// TwinCAT 3 PLC project PayloadCarrier
// ProgramVersion: 3.1.4023.0
// libraries:
//   Tc2_Standard, * (Beckhoff Automation GmbH)
//   Tc2_System, * (Beckhoff Automation GmbH)
//   Tc3_Module, * (Beckhoff Automation GmbH)
// project tree:
//   DUTs/ E_PAYLOAD_CARRIER_MODE.TcDUT, E_Payload_Type.TcDUT, ST_SynchPayload.TcDUT
//   GVLs/ Global.TcGVL
//   / PlcTask.TcTTO
//   POUs/ A_Payload.TcPOU, I_Payload.TcIO, I_Payload_A.TcIO, I_Payload_B.TcIO, PayloadCarrier.TcPOU, Payload_A.TcPOU, MAIN.TcPOU, Payload_B.TcPOU, StepChain_1.TcPOU, StepChain_2.TcPOU, SynchPayload.TcPOU
// real-time tasks:
//   TASK PlcTask: cycle T#10ms, priority 20, ADS port 350

CONFIGURATION PayloadCarrier
    RESOURCE PLC ON TwinCAT3
        TASK PlcTask(INTERVAL := T#10ms, PRIORITY := 20);
        PROGRAM MAIN WITH PlcTask : MAIN;
    END_RESOURCE
END_CONFIGURATION

// ---- DUTs/E_PAYLOAD_CARRIER_MODE.TcDUT
TYPE E_PAYLOAD_CARRIER_MODE :
(
	NO_PAYLOAD_CARRIER_MODE := 0,
	ONE_TO_ONE := 10,
	ONE_TO_MANY := 15,
	SHARED := 50,
	RESTRICTED := 55
);
END_TYPE

// ---- DUTs/E_Payload_Type.TcDUT

TYPE E_Payload_Type :
(
	NO_PAYLOAD := 0,
	PAYLOAD_A,
	PAYLOAD_B,
	SYNCH_PAYLOAD,
	PAYLOAD_TYPE_SIZE
);
END_TYPE

// ---- DUTs/ST_SynchPayload.TcDUT
TYPE ST_SynchPayload :
STRUCT
	bReleaseRequest : BOOL;
	bReleaseRequestReceived : BOOL;
	bRequestAck : BOOL;
	bRequestAckReceived : BOOL;
END_STRUCT
END_TYPE

// ---- GVLs/Global.TcGVL
VAR_GLOBAL
	fbPayloadCarrier : PayloadCarrier;
END_VAR

// ---- POUs/I_Payload.TcIO
INTERFACE I_Payload EXTENDS __System.IQueryInterface

END_INTERFACE

// ---- POUs/I_Payload_A.TcIO
INTERFACE I_Payload_A EXTENDS I_Payload

END_INTERFACE

// ---- POUs/I_Payload_B.TcIO
INTERFACE I_Payload_B EXTENDS I_Payload

END_INTERFACE

// ---- POUs/MAIN.TcPOU
PROGRAM MAIN
VAR
	
	fbStepChain_1 : StepChain_1;
	fbStepChain_2 : StepChain_2;
	
	fbPayloadA : Payload_A;
	pPayloadA : POINTER TO Payload_A;
	fbPayloadB : Payload_B;
	
	rPayloadAReceiver : REFERENCE TO Payload_A;
	pPayloadAReceiver : POINTER TO Payload_A;
	fbPayloadAReceiver : Payload_A;
	pPayloadBReceiver : POINTER TO Payload_B;
	iPayload : I_Payload;
	step : INT;
	
END_VAR

fbPayloadCarrier();
//fbPayloadA();
//fbPayloadB();

fbStepChain_1();
fbStepChain_2();

(*
CASE step OF
	
	1:
	
		IF 	fbPayloadCarrier.SetPayload(fbPayloadA,PAYLOAD_A,ONE_TO_ONE)
			THEN
			
			step := 2;
		END_IF
		
	2:
	
		IF	fbPayloadCarrier.GetPayload(pPayloadAReceiver,PAYLOAD_A)
			THEN
			
			step := 3;
		END_IF
		
	3:
	
	4:

		fbPayloadCarrier.ResetPayload();
		
	10:
	
		pPayloadA := __NEW(PAYLOAD_A);
		IF 	fbPayloadCarrier.SetPayload(pPayloadA^,PAYLOAD_A,ONE_TO_ONE)
			THEN
			
			step := 11;
		END_IF
		
	11:
	
		IF	fbPayloadCarrier.GetPayload(pPayloadAReceiver,PAYLOAD_A)
			THEN
			
			step := 12;
		END_IF
		
	12:
	
	13:
	
		__DELETE(pPayloadA);
		step := 14;
		
	14:
		
	15:

		fbPayloadCarrier.ResetPayload();	
		
END_CASE
*)

END_PROGRAM

// ---- POUs/StepChain_1.TcPOU
FUNCTION_BLOCK StepChain_1
VAR_INPUT
END_VAR
VAR_OUTPUT
END_VAR
VAR
	fbSynchPayload : SynchPayload;
	step : UINT;
END_VAR

CASE step OF
	
	0:
		IF 	fbPayloadCarrier
				.SetPayload(
					fbSynchPayload,
					SYNCH_PAYLOAD,
					ONE_TO_ONE,
					THIS
				)	
			THEN
			
			step := 10;
		END_IF
		
	10:
	
		fbSynchPayload.bReleaseRequest := TRUE;
		IF 	fbSynchPayload.bReleaseRequestReceived
			THEN
			fbSynchPayload.bReleaseRequest := FALSE;
			step := 20;
		END_IF
		
	20:
		IF  fbSynchPayload.bRequestAck
			THEN
			fbSynchPayload.bRequestAckReceived := TRUE;
			step := 30;
		END_IF
		
	30:	

		fbSynchPayload.bRequestAckReceived := FALSE;
		step := 40;
		
	40:
	
		fbPayloadCarrier.ResetPayload(THIS);
		step := 50;
		
		
END_CASE

END_FUNCTION_BLOCK

// ---- POUs/SynchPayload.TcPOU
FUNCTION_BLOCK SynchPayload IMPLEMENTS I_Payload
VAR_INPUT
	bReleaseRequest : BOOL;
	bReleaseRequestReceived : BOOL;
	bRequestAck : BOOL;
	bRequestAckReceived : BOOL;
END_VAR
VAR_OUTPUT
END_VAR
VAR
END_VAR

END_FUNCTION_BLOCK

// ---- POUs/StepChain_2.TcPOU
FUNCTION_BLOCK StepChain_2
VAR_INPUT
END_VAR
VAR_OUTPUT
END_VAR
VAR
	pSynchPayload : POINTER TO SynchPayload;
	step : UINT;
	timer : TON;
END_VAR

timer(PT:= T#4S);
IF 	pSynchPayload = 0
	THEN
	
	step := 0;
END_IF

CASE step OF
	
	0:
		IF 	fbPayloadCarrier.GetPayload(pSynchPayload,SYNCH_PAYLOAD)
			THEN
			
			step := 10;
		END_IF
		
	10:
	
		IF 	pSynchPayload^.bReleaseRequest
			THEN
			
			pSynchPayload^.bReleaseRequestReceived := TRUE;
			step := 20;
		END_IF
		
	20:
		pSynchPayload^.bReleaseRequestReceived := FALSE;
		timer.IN := TRUE;
		IF  timer.Q
			THEN
			timer.IN := FALSE;
			pSynchPayload^.bRequestAck := TRUE;
			step := 30;
		END_IF
		
	30:	

		IF 	pSynchPayload^.bRequestAckReceived
			THEN
			pSynchPayload^.bRequestAck := FALSE;
			step := 40;
		END_IF
	
	40:;
		
		
END_CASE

END_FUNCTION_BLOCK

// ---- POUs/Payload_A.TcPOU
{attribute 'enable_dynamic_creation'}
FUNCTION_BLOCK Payload_A IMPLEMENTS I_Payload_A
VAR_INPUT
END_VAR
VAR_OUTPUT
END_VAR
VAR
	nPayload : INT;
END_VAR

END_FUNCTION_BLOCK

// ---- POUs/Payload_B.TcPOU
FUNCTION_BLOCK Payload_B IMPLEMENTS I_Payload_B
VAR_INPUT
END_VAR
VAR_OUTPUT
END_VAR
VAR
	bPayload : BOOL;
END_VAR

END_FUNCTION_BLOCK

// ---- POUs/PayloadCarrier.TcPOU
FUNCTION_BLOCK PayloadCarrier 
VAR_INPUT
END_VAR
VAR_OUTPUT
END_VAR
VAR
	//aPayloads : ARRAY[1..PAYLOAD_TYPE_SIZE-1] OF I_Payload;
	iPayload : I_Payload;
	ePayloadType : E_Payload_Type;
	aGarbageCollection : ARRAY[1..cSizeOfGarbageCollection] OF POINTER TO POINTER TO BYTE;
	nGarbageCollectionCounter : UINT;
	bLock : BOOL;
	bPayloadAssigned : BOOL;
	ePayloadCarrierMode : E_PAYLOAD_CARRIER_MODE;
	pResetKey : POINTER TO BYTE;
END_VAR
VAR CONSTANT
	cSizeOfGarbageCollection : UINT := 10 * ( PAYLOAD_TYPE_SIZE-1 );
END_VAR

METHOD GetPayload : BOOL
VAR_IN_OUT
	pByte : POINTER TO BYTE;
END_VAR

VAR_INPUT
	ePayloadType : E_Payload_Type;
END_VAR
(*
IF 	THIS^.ePayloadType = ePayloadType
	THEN
		GetPayload :=  __QUERYPOINTER(iPayload, pByte);
END_IF
*)


IF 	iPayload <> 0(*aPayloads[ePayloadType] <> 0*)
	AND THIS^.ePayloadType = ePayloadType
	AND nGarbageCollectionCounter <= cSizeOfGarbageCollection
	AND (
			ePayloadCarrierMode = ONE_TO_MANY
			OR 
			(
				ePayloadCarrierMode = ONE_TO_ONE 
				AND NOT bPayloadAssigned
			)
		)
	THEN
	
		bPayloadAssigned := (ePayloadCarrierMode = ONE_TO_ONE); 
		GetPayload :=   __QUERYPOINTER(iPayload , pByte);// __QUERYPOINTER(aPayloads[ePayloadType], pByte);
		IF 	GetPayload
			THEN
			
			nGarbageCollectionCounter := nGarbageCollectionCounter + 1;
			aGarbageCollection[nGarbageCollectionCounter] := ADR(pByte);
			
		END_IF
		
END_IF
END_METHOD

METHOD ResetPayload : BOOL
VAR_INPUT
	pResetKey : POINTER TO BYTE;
END_VAR
VAR
	i: UINT;
END_VAR
IF 	nGarbageCollectionCounter > 0
	AND pResetKey = THIS^.pResetKey
	THEN
	
	FOR i := 1 TO nGarbageCollectionCounter DO
		aGarbageCollection[i]^ := 0;	
		aGarbageCollection[i]:= 0;		
	END_FOR
	
	nGarbageCollectionCounter := 0;
	(*
	FOR i := 1 TO PAYLOAD_TYPE_SIZE-1 DO
		aPayloads[i] := 0;
	END_FOR
	*)
	iPayload := 0;
	bPayloadAssigned := FALSE;
	bLock := FALSE;
	ResetPayload := TRUE;
	
END_IF
END_METHOD

METHOD SetPayload : BOOL
VAR_INPUT
	iPayload : I_Payload; 
	ePayloadType : E_Payload_Type;
	ePayloadCarrierMode : E_PAYLOAD_CARRIER_MODE;
	pResetKey : POINTER TO BYTE;
END_VAR
(*
IF ePayloadType <> NO_PAYLOAD
	THEN
	
	THIS^.iPayload := iPayload;
	THIS^.ePayloadType := ePayloadType;
	
	SetPayload := TRUE;
	
END_IF
*)

IF 	ePayloadType <> NO_PAYLOAD
	AND ePayloadCarrierMode <> NO_PAYLOAD_CARRIER_MODE
	AND bLock = FALSE
	AND pResetKey <> 0
	THEN
	
	this^.pResetKey := pResetKey;
	bLock := TRUE;
	
	THIS^.ePayloadCarrierMode := ePayloadCarrierMode;
	//THIS^.aPayloads[ePayloadType] := iPayload;
	THIS^.iPayload := iPayload;
	THIS^.ePayloadType := ePayloadType;
	SetPayload := TRUE;
	
END_IF
END_METHOD

END_FUNCTION_BLOCK

// ---- POUs/A_Payload.TcPOU
FUNCTION_BLOCK ABSTRACT A_Payload
VAR_INPUT
END_VAR
VAR_OUTPUT
END_VAR
VAR
END_VAR

END_FUNCTION_BLOCK
